TYPE T_OnlineChangeTestRuntime :
STRUCT
	nMainCycles: UDINT;
	nTotalPanic: UDINT;
	nTotalWarn: UDINT;
END_STRUCT
END_TYPE

(* stored: Version 1.1.0.1
   DUT T_OnlineChangeTestRuntime: Id {5acbe042-8503-4011-ba67-2e24f766cfa8} *)
